FUNCTION_BLOCK MLMODELSIM (* Module that simulates the operation of an ML model for adjusting values for regulators *)
  (* Version 1.0, AN, SWDC RTSoft *)
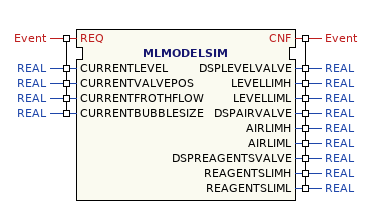
  EVENT_INPUT
    REQ WITH CURRENTLEVEL, CURRENTVALVEPOS, CURRENTFROTHFLOW, CURRENTBUBBLESIZE;
  END_EVENT
  EVENT_OUTPUT
    CNF WITH DSPLEVELVALVE, LEVELLIMH, LEVELLIML, DSPAIRVALVE, AIRLIMH, AIRLIML, DSPREAGENTSVALVE, REAGENTSLIMH, REAGENTSLIML;
  END_EVENT
  VAR_INPUT
    CURRENTLEVEL : REAL;
    CURRENTVALVEPOS : REAL;
    CURRENTFROTHFLOW : REAL;
    CURRENTBUBBLESIZE : REAL;
  END_VAR
  VAR_OUTPUT
    DSPLEVELVALVE : REAL;
    LEVELLIMH : REAL;
    LEVELLIML : REAL;
    DSPAIRVALVE : REAL;
    AIRLIMH : REAL;
    AIRLIML : REAL;
    DSPREAGENTSVALVE : REAL;
    REAGENTSLIMH : REAL;
    REAGENTSLIML : REAL;
  END_VAR
END_FUNCTION_BLOCK
